PROGRAM MAIN
VAR
END_VAR

END_PROGRAM

(* stored: Version 1.1.0.1
   POU MAIN: Id {f0184b22-5e3f-456c-8816-e294e8130996} *)
